Staubli VAL3: getErrorMessage.pgx

public program getErrorMessage(string& x_sMessage[] (dimensions=1))
begin
  // This programs returns a clear text about the last error code
  //
  // Input Param
  // None
  //
  // Output Param
  //  x_sMessage    : Error message
  //
  //--------------------------------------------------------------
  //
  x_sMessage=sErrorMessage
end
